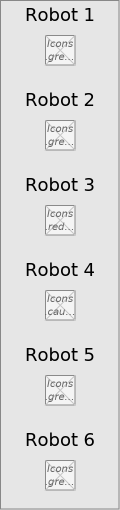
VISUALIZATION LeftRobotStatus  // 120x510
    Textfield (0,0 120x30), "Robot 1"
    Textfield (0,85 120x30), "Robot 2"
    Textfield (0,170 120x30), "Robot 3"
    Textfield (0,255 120x30), "Robot 4"
        OnMouseClick: execute { UI.FrameSelector.SelectedFrame := 1; }
    Textfield (0,340 120x30), "Robot 5"
    Textfield (0,425 120x30), "Robot 6"
    Image (45,35 30x30), input disabled if: TRUE, image: Icons.green-checkmark-icon
    Image (45,120 30x30), image: Icons.green-checkmark-icon
    Image (45,205 30x30), image: Icons.red-x-icon
    Image (45,290 30x30), image: Icons.caution-icon
        OnMouseClick: execute { UI.FrameSelector.SelectedFrame := 1; }
    Image (45,375 30x30), image: Icons.green-checkmark-icon
    Image (45,460 30x30), image: Icons.green-checkmark-icon
END_VISUALIZATION

(* stored: Version 1.1.0.1, ProductVersion 3.1.4024.15
   Visu LeftRobotStatus: Id {6529ba2d-709b-40cb-a5a1-3ee826275302} *)
